// TwinCAT 3 PLC project Main
// ProgramVersion: 3.1.4023.0
// libraries:
//   Tc2_Standard, * (Beckhoff Automation GmbH)
//   Tc2_System, * (Beckhoff Automation GmbH)
//   Tc2_Utilities, * (Beckhoff Automation GmbH)
//   Tc3_Module, * (Beckhoff Automation GmbH)
// project tree:
//   DUTs/ tDriveInNState1.TcDUT (not stored), tDriveInNState2.TcDUT, tDriveOutNCtrl1.TcDUT, tEncInState1.TcDUT (not stored), tEncInState2.TcDUT (not stored), tEncOutNCtrl1.TcDUT (not stored)
//   / PlcTask.TcTTO (not stored)
//   POUs/ MAIN.TcPOU
// real-time tasks:
//   TASK PlcTask: cycle T#10ms, priority 20, ADS port 350
// motion (NC):
//   TASK NC-Task 1 SAF: cycle T#2ms, priority 4, ADS port 501
//   TASK NC-Task 1 SVB: cycle T#10ms, priority 8, ADS port 511
//   AXIS ConveyorMotorAxis (id 1)
//     Dynamic: AccelerationMaximum=50, DecelerationMaximum=50, Acceleration=29.9999, Deceleration=29.9999, Jerk=44.9998
//     Velo: SlowManual=10, FastManual=30, Maximum=30
//     OtherSettings: AllowMotionCmdToSlave=true
//     encoder EncType=4
//       EncPara: MaxCount=#x0000ffff
//         Inc: RefSoftSyncMask=#x0000ffff
//     drive DrvType=23
//       Analog: VeloReferenz=30, TorqueSetpointScale=10, ScaleFactorActTorque=0.1
//       TimeComp: TaskDelayCycles=1
//     controller CtrType=1
//       CtrPara: PriorControlFactor=1
//         PosDiffControl: Enable=false
//         Observer: BandWidth=20
//   AXIS Achse 2 (id 2)
//     OtherSettings: AllowMotionCmdToSlave=true
//     encoder EncType=4
//       EncPara: MaxCount=#x0000ffff
//         Inc: RefSoftSyncMask=#x0000ffff
//     drive DrvType=23
//       Analog: TorqueSetpointScale=10, ScaleFactorActTorque=0.1
//       TimeComp: TaskDelayCycles=1
//     controller CtrType=1
//       CtrPara: PriorControlFactor=1
//         Observer: BandWidth=20
// I/O:
//   DEVICE Gerät 1 (EtherCAT) (disabled), AmsNetId 192.168.8.155.2.1
//     Klemme 1 (EK1100) [EK1100 EtherCAT-Koppler (2A E-Bus)]
//       Klemme 2 (EL7342) [EL7342 2K. DC-Motor-Endstufe (50V, 3.5A)]
// variable links:
//   NC-Task 1 SAF/Axes/Achse 2 <-> Device 1 (EtherCAT)/Term 1 (EK1100)/Term 2 (EL7342)
//     Drive/Inputs/In/nState1 @bit 3 <-> DCM Status Channel 1/Status/Error
//     Drive/Inputs/In/nState1 @bit 5 <-> DCM Status Channel 1/Status/Moving negative
//     Drive/Inputs/In/nState1 @bit 4 <-> DCM Status Channel 1/Status/Moving positive
//     Drive/Inputs/In/nState1 @bit 1 <-> DCM Status Channel 1/Status/Ready
//     Drive/Inputs/In/nState1 <-> DCM Status Channel 1/Status/Ready to enable
//     Drive/Inputs/In/nState1 @bit 6 <-> DCM Status Channel 1/Status/Torque reduced
//     Drive/Inputs/In/nState1 @bit 2 <-> DCM Status Channel 1/Status/Warning
//     Drive/Inputs/In/nState2 @bit 3 <-> DCM Status Channel 1/Status/Digital input 1
//     Drive/Inputs/In/nState2 @bit 4 <-> DCM Status Channel 1/Status/Digital input 2
//     Drive/Inputs/In/nState2 @bit 5 <-> DCM Status Channel 1/Status/Sync error
//     Drive/Inputs/In/nState2 @bit 7 <-> DCM Status Channel 1/Status/TxPDO Toggle
//     Drive/Inputs/In/nState4 @bit 1 <-> WcState/InputToggle
//     Drive/Inputs/In/nState4 <-> WcState/WcState
//     Drive/Outputs/Out/nCtrl1 <-> DCM Control Channel 1/Control/Enable
//     Drive/Outputs/Out/nCtrl1 @bit 2 <-> DCM Control Channel 1/Control/Reduce torque
//     Drive/Outputs/Out/nCtrl1 @bit 1 <-> DCM Control Channel 1/Control/Reset
//     Drive/Outputs/Out/nCtrl1 @bit 3 <-> DCM Control Channel 1/Control/Threshold active
//     Drive/Outputs/Out/nDataOut2[0] <-> DCM Velocity Channel 1/Velocity
//     Enc/Inputs/In/nDataIn1[0] <-> ENC Status compact Channel 1/Counter value
//     Enc/Inputs/In/nDataIn2[0] <-> ENC Status compact Channel 1/Latch value
//     Enc/Inputs/In/nState1 @bit 4 <-> ENC Status compact Channel 1/Status/Counter overflow
//     Enc/Inputs/In/nState1 @bit 3 <-> ENC Status compact Channel 1/Status/Counter underflow
//     Enc/Inputs/In/nState1 @bit 7 <-> ENC Status compact Channel 1/Status/Extrapolation stall
//     Enc/Inputs/In/nState1 @bit 1 <-> ENC Status compact Channel 1/Status/Latch extern valid
//     Enc/Inputs/In/nState1 @bit 2 <-> ENC Status compact Channel 1/Status/Set counter done
//     Enc/Inputs/In/nState2 @bit 4 <-> ENC Status compact Channel 1/Status/Status of extern latch
//     Enc/Inputs/In/nState2 <-> ENC Status compact Channel 1/Status/Status of input A
//     Enc/Inputs/In/nState2 @bit 1 <-> ENC Status compact Channel 1/Status/Status of input B
//     Enc/Inputs/In/nState2 @bit 5 <-> ENC Status compact Channel 1/Status/Sync error
//     Enc/Inputs/In/nState2 @bit 7 <-> ENC Status compact Channel 1/Status/TxPDO Toggle
//     Enc/Inputs/In/nState4 @bit 1 <-> WcState/InputToggle
//     Enc/Inputs/In/nState4 <-> WcState/WcState
//     Enc/Outputs/Out/nCtrl1 @bit 3 <-> ENC Control compact Channel 1/Control/Enable latch extern on negative edge
//     Enc/Outputs/Out/nCtrl1 @bit 1 <-> ENC Control compact Channel 1/Control/Enable latch extern on positive edge
//     Enc/Outputs/Out/nCtrl1 @bit 2 <-> ENC Control compact Channel 1/Control/Set counter
//     Enc/Outputs/Out/nDataOut1[0] <-> ENC Control compact Channel 1/Set counter value
//   Main/Main Instance <-> NC-Task 1 SAF/Axes/ConveyorMotorAxis
//     PlcTask Inputs/MAIN.velocity <-> Drive/Outputs/Out/nDataOut2[0]
//     PlcTask Outputs/MAIN.counterValue <-> Enc/Inputs/In/nDataIn1[0]
//     PlcTask Outputs/MAIN.driveInState1 <-> Drive/Inputs/In/nState1

// ---- DUTs/tDriveInNState2.TcDUT
TYPE tDriveInNState2 :
STRUCT
	DigitalInput1	: BIT;
	DigitalInput2	: BIT;
	SyncError		: BIT;
	TcPdoToggle		: BIT;
END_STRUCT
END_TYPE

// ---- DUTs/tDriveOutNCtrl1.TcDUT
TYPE tDriveOutNCtrl1 :
STRUCT
	Enable			: BIT;
	Reset			: BIT;
	ReduceTorque	: BIT;
	ThresholdActive	: BIT;
END_STRUCT
END_TYPE

// ---- POUs/MAIN.TcPOU
PROGRAM MAIN
VAR
	velocity		AT%I*	: INT;		// nDataOut2[0] . nDataOut2 . Out . Ausgänge . Drive . ConveyorMotorAxis . ConveyorMotorAxis . Achsen . NC-Task 1 SAF
	counterValue 	AT%Q*	: UINT := 0;		//nDataIn1[0] . nDataIn1 . In . Eingänge . Enc . ConveyorMotorAxis . ConveyorMotorAxis . Achsen . NC-Task 1 SAF
	driveInState1	AT%Q*	: USINT;	// State of the hardware motor module
	
	
	ModelToPLC		: DWORD := 0;		// empty (1), driveInState1 (1), counterValue (2)
	PLCToModel		: DWORD := 0;		// empty (2), velocity (2)
END_VAR

// Communication
// ToPlc
counterValue := DWORD_TO_UINT(ModelToPLC AND 16#00_00_FF_FF);
driveInState1 := DWORD_TO_USINT(SHR((ModelToPLC AND 16#00_FF_00_00),16));


// ToModel
PLCToModel := 0;
PLCToModel := SHL((PLCToModel OR velocity),0);

END_PROGRAM
